// TIA Portal V20 export
TYPE "LER_typeCommunicationData_Conveyor"
// stored: Access Published
   STRUCT
      UnitStatus : "LER_typeCommunicationUnitStatus";
      InterfaceData : "LER_typeCommunicationInterfaceData";
   END_STRUCT;
END_TYPE
